{attribute 'no_explicit_call' := 'Do not call the body - Stick to OOP'}
// Check zone start to end in positive direktion.
FUNCTION_BLOCK FB_XP_Zone EXTENDS FB_CH_Object IMPLEMENTS I_XP_Zone
VAR
	{attribute 'hide'}
	bInitDone : BOOL;
	{attribute 'hide'}
	ipXpSystem : I_XP_System_Registration; //Interface to XPlanar system 
	{attribute 'hide'}
	ipListOfMoversToCheck : CHALET_BaseComponents.I_CH_LIST;
	{attribute 'hide'}
	aMoversInZone : ARRAY [0..(CHALET_BaseComponents.BaseParameterlist.MAX_OBJECTS-1)] OF I_XP_Mover_PLC;
	{attribute 'hide'}
	fStartPositionOnTrack : LREAL;
	{attribute 'hide'}
	fEndPositionOnTrack : LREAL;	
	{attribute 'hide'}
	ipAccocietedTrack : I_XP_Track;
END_VAR

{attribute 'monitoring':='call'}
PROPERTY AccocietedTrack : I_XP_Track
GET
AccocietedTrack := THIS^.ipAccocietedTrack;
END_GET
SET
THIS^.ipAccocietedTrack := AccocietedTrack;
END_SET
END_PROPERTY

{attribute 'monitoring':='call'}
PROPERTY CtsMoversInZone : UINT
GET
VAR
	nIndex : UDINT;
END_VAR
THIS^.Prepare();//Prepare Time-critical information

//Check array for entrys, exit if fisrt empty arrayindex is found.
FOR nIndex := 0 TO (CHALET_BaseComponents.BaseParameterlist.MAX_OBJECTS-1) DO
	IF (aMoversInZone[nIndex] <> 0) THEN
		CtsMoversInZone := CtsMoversInZone +1;
	ELSE
		RETURN;
	END_IF
END_FOR
END_GET
END_PROPERTY

{attribute 'monitoring':='call'}
PROPERTY EndPositionOnTrack : LREAL
GET
EndPositionOnTrack := fEndPositionOnTrack;
END_GET
SET
fEndPositionOnTrack := EndPositionOnTrack;
END_SET
END_PROPERTY

METHOD FB_init : BOOL
VAR_INPUT
	bInitRetains : BOOL; // if TRUE, the retain variables are initialized (warm start / cold start)
	bInCopyCode : BOOL;  // if TRUE, the instance afterwards gets moved into the copy code (online change)
	
	ipXpSystem : I_XP_System_Registration; //Interface to XPlanar system object
END_VAR
VAR_INST
	{attribute 'hide'}
	bFBInitCalledOnce : BOOL; //Do the following code once during start up and not during onlinechange
END_VAR
//Do the following code once during start up and not during onlinechange
IF NOT bFBInitCalledOnce THEN 
	;
END_IF

//Regristrate object in System if unknown
IF ipXpSystem <> 0 AND THIS^.ipXpSystem = 0 THEN
	ipXpSystem.RegisterZone(THIS^);
	THIS^.ipXpSystem := ipXpSystem;
END_IF

bFBInitCalledOnce := TRUE;
END_METHOD

{attribute 'monitoring':='call'}
PROPERTY HR : HRESULT
GET
IF ipAccocietedTrack <> 0 AND_THEN ipAccocietedTrack.Length > 0 THEN
	HR := S_OK;
ELSE
	HR := E_FAIL;
END_IF
END_GET
END_PROPERTY

METHOD Initialize : HRESULT
IF THIS^.ipXpSystem = 0 THEN
	//No valide interface
	Initialize := E_FAIL;
	RETURN;
END_IF


IF (THIS^.ipListOfMoversToCheck <> 0) AND (THIS^.ipAccocietedTrack <> 0) THEN
	THIS^.bInitDone := TRUE;
	Initialize := S_OK;
ELSE
	Initialize := E_FAIL;
END_IF
END_METHOD

PROPERTY ListOfMoversToCheck : I_CH_List
SET
IF ListOfMoversToCheck <> 0 THEN
	ipListOfMoversToCheck := ListOfMoversToCheck;
END_IF
END_SET
END_PROPERTY

{attribute 'monitoring':='call'}
PROPERTY MoversInZone : REFERENCE TO ARRAY [0..(CHALET_BaseComponents.BaseParameterlist.MAX_OBJECTS-1)] OF I_XP_Mover_PLC // Return a sorted list of movers in this zone. Index 0 is the mover in Front.
GET
THIS^.Prepare();//Prepare Time-critical information

MoversInZone REF= THIS^.aMoversInZone;
END_GET
END_PROPERTY

(* Time-critical information is processed here, which can then be polled via the property every cycle. 
The update method is usually at the end of the program and then it is already 'outdated'. *)
METHOD PRIVATE Prepare : HRESULT
VAR
	nLoopIndex : UDINT;
	ipMoverPlc : I_XP_Mover_PLC;
	fDistToStart : LREAL;
	aDisanceToStart : ARRAY [0..(CHALET_BaseComponents.BaseParameterlist.MAX_OBJECTS-1)] OF LREAL;
END_VAR
VAR_INST
	{attribute 'hide'}
	nLastUpdatedCycleCount : UDINT;
END_VAR
//Check if this Cycle the dates are allready prepared
IF nLastUpdatedCycleCount <> TwinCAT_SystemInfoVarList._TaskInfo[THIS^.nTaskIndex].CycleCount THEN
	nLastUpdatedCycleCount := TwinCAT_SystemInfoVarList._TaskInfo[THIS^.nTaskIndex].CycleCount;

	//Clear array
	MEMSET(destAddr:=ADR(aMoversInZone),n:=SIZEOF(aMoversInZone),fillByte:=0);
	
	//Cheack all Movers and generate a sorted list of all mover in this zone
	THIS^.ipListOfMoversToCheck.ResetIterator();
	WHILE THIS^.ipListOfMoversToCheck.HasNextObject() DO
		IF __QUERYINTERFACE(THIS^.ipListOfMoversToCheck.GetNextObject(),ipMoverPlc) THEN
			
			//If in zone
			IF ipMoverPlc.CurrentTrack = THIS^.ipAccocietedTrack AND_THEN (fStartPositionOnTrack <= ipMoverPlc.PositionOnTrack) AND (fEndPositionOnTrack >= ipMoverPlc.PositionOnTrack) AND (fStartPositionOnTrack <= fEndPositionOnTrack) THEN
				fDistToStart := fEndPositionOnTrack - ipMoverPlc.PositionOnTrack;
				
				//Check array of movers and decide if the current one is closer to 
				FOR nLoopIndex := 0 TO (CHALET_BaseComponents.BaseParameterlist.MAX_OBJECTS-1) DO
					//empty array position
					IF aMoversInZone[nLoopIndex] = 0 THEN
						aMoversInZone[nLoopIndex] := ipMoverPlc;
						aDisanceToStart[nLoopIndex] := fDistToStart;
						EXIT;
						
					//Closer Mover found, move whole array 	
					ELSIF aDisanceToStart[nLoopIndex] > fDistToStart THEN
						MEMMOVE(srcAddr := ADR(aMoversInZone[nLoopIndex]), destAddr := ADR(aMoversInZone[nLoopIndex+1]), n := (SIZEOF(aMoversInZone[0])*(CHALET_BaseComponents.BaseParameterlist.MAX_OBJECTS-1)));
						MEMMOVE(srcAddr := ADR(aDisanceToStart[nLoopIndex]), destAddr := ADR(aDisanceToStart[nLoopIndex+1]), n := (SIZEOF(aDisanceToStart[0])*(CHALET_BaseComponents.BaseParameterlist.MAX_OBJECTS-1)));
						aMoversInZone[nLoopIndex] := ipMoverPlc;
						aDisanceToStart[nLoopIndex] := fDistToStart;
						EXIT;
						
					//check next position	
					ELSE 
						;
					END_IF
				END_FOR
			END_IF
		END_IF
	END_WHILE
END_IF
END_METHOD

{attribute 'monitoring':='call'}
PROPERTY StartPositionOnTrack : LREAL
GET
StartPositionOnTrack := fStartPositionOnTrack;
END_GET
SET
fStartPositionOnTrack := StartPositionOnTrack;
END_SET
END_PROPERTY

METHOD Update : HRESULT
VAR

END_VAR
// Nothing todo in Update. Check Prepare
END_METHOD

END_FUNCTION_BLOCK

(* stored: Version 1.1.0.1, ProductVersion 3.1.4024.12
   POU FB_XP_Zone: Id {9b5c2aba-5d65-4390-8f35-cbd4e5d75462}, SpecialFunc None
   Property AccocietedTrack: Id {54f95ac3-51d8-4f2e-bb9d-69155c8c8898}
   Get Get: Id {2aec8e3b-a953-4173-b2ba-5286050316b3}
   Set Set: Id {2eca0fca-089c-4144-85b7-ed68c2ecb24c}
   Property CtsMoversInZone: Id {5fcab65a-c45f-48aa-9861-8c583938c821}
   Get Get: Id {8b39be2e-11bb-4852-a3c8-d4c2357f42e8}
   Property EndPositionOnTrack: Id {a0fa287d-9b0c-40ab-838b-6912a44e3896}
   Get Get: Id {0748fc3f-261f-46af-95b0-f775d75211bf}
   Set Set: Id {c09dcc01-0559-4021-a6a5-2ce84419f470}
   Method FB_init: Id {6e983b48-77a3-4dff-900b-b1bd15863c70}
   Property HR: Id {a14fee94-3257-4d49-8f83-cbcb4fe15ef7}
   Get Get: Id {3ecbfe86-e365-4eb3-b9a3-44450e89b85a}
   Method Initialize: Id {bded9a3f-15e5-4382-a88c-b201de005416}
   Property ListOfMoversToCheck: Id {857ff228-6ee0-43a7-8a6a-1db86eb1fb2c}
   Set Set: Id {a4c5f319-273f-405f-aa39-ac407eb7a61e}
   Property MoversInZone: Id {d637c274-a77a-4857-a4ee-3f4555864a74}
   Get Get: Id {8409ff4e-605e-4576-a1bf-903a1943eced}
   Method Prepare: Id {f7cecc17-4d6f-4b63-bc01-d1776bce3f38}
   Property StartPositionOnTrack: Id {db42354e-ef45-425c-b30c-a2d6abbf207d}
   Get Get: Id {14b70797-8a1a-45b4-946c-8aba3c90796d}
   Set Set: Id {137f1219-958d-4a1d-b795-cab82da4b5eb}
   Method Update: Id {a57b36be-57e2-46fb-ac48-3faaf13c289d} *)
